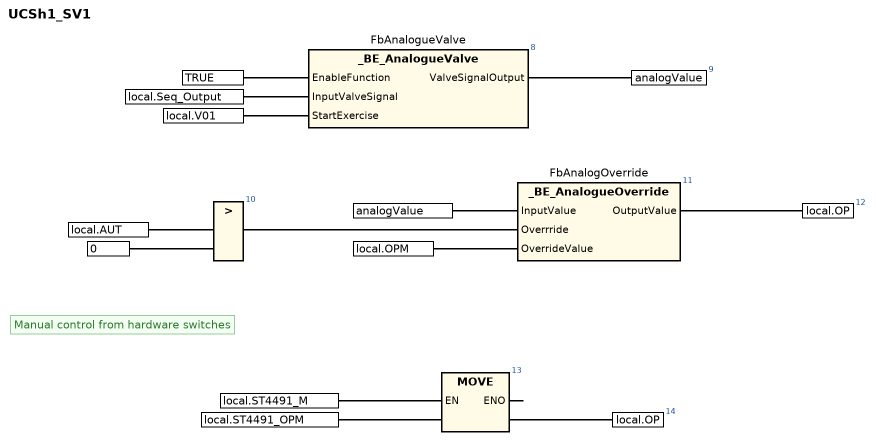
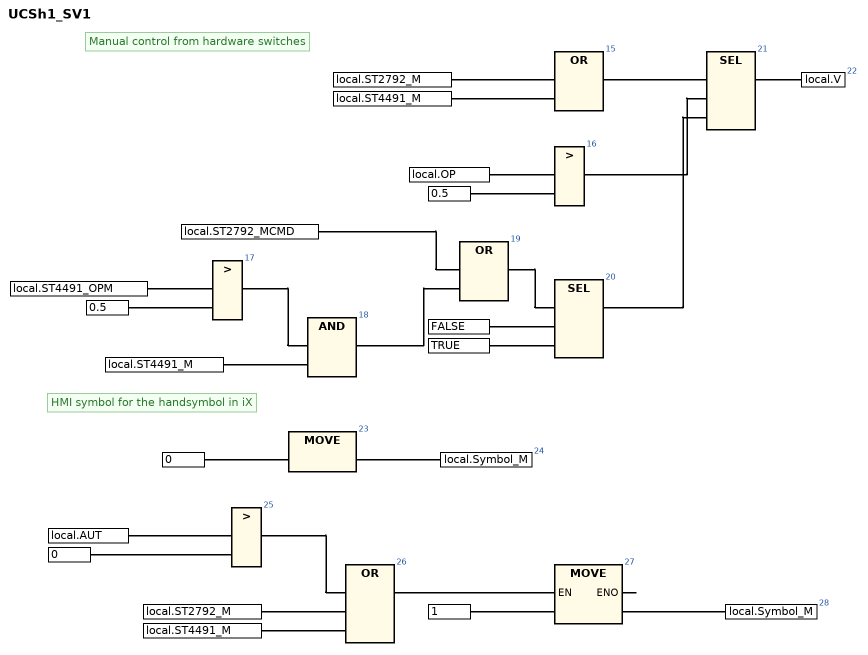
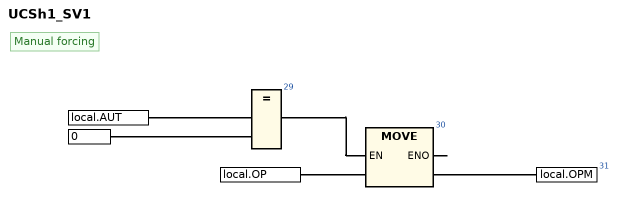
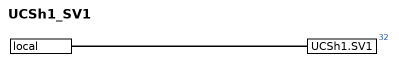
UCSh1.SV1.Seq_Output := UCSh1.GT1.OP;
local := UCSh1.SV1;
fbExercise(
    EnableFunction := local.Ex_En,
    RunIndication := local.OP > 0.5,
    DaysBetweenExercise := local.SP1,
    HoursBetweenExercise := local.SP2,
    EnableDay := local.Ex_En_Day,
    ExerciseStartDay := local.SP3,
    EnableHourMinute := local.Ex_En_Time,
    ExerciseStartHour := local.SP4,
    ExerciseStartMinute := local.SP5,
    ExerciseRunTime := local.SP6,
    SecondPulse := SYS_SecondPulse,
    ClockArray := SYS_ArrayPlcTime,
    SecondsIncObjectOff := local.Ex_SecOff,
    SavedWorkingData := local.Ex_SavedData); // _BE_Exercise
local.V01 := fbExercise.ExerciseActive;
local.PV1 := fbExercise.DaysLeft;
local.PV2 := fbExercise.HoursLeft;
local.PV3 := fbExercise.MinutesLeft;
FbAnalogueValve(EnableFunction := TRUE, InputValveSignal := local.Seq_Output, StartExercise := local.V01); // _BE_AnalogueValve
analogValue := FbAnalogueValve.ValveSignalOutput;
FbAnalogOverride(InputValue := analogValue, Overrride := local.AUT > 0, OverrideValue := local.OPM); // _BE_AnalogueOverride
local.OP := FbAnalogOverride.OutputValue;
// Manual control from hardware switches
IF local.ST4491_M THEN _w1 := local.ST4491_OPM; END_IF
local.OP := _w1;
// Manual control from hardware switches
local.V := SEL(local.ST2792_M OR local.ST4491_M, local.OP > 0.5, SEL(local.ST2792_MCMD OR local.ST4491_OPM > 0.5 AND local.ST4491_M, FALSE, TRUE));
// HMI symbol for the handsymbol in iX
local.Symbol_M := 0;
IF local.AUT > 0 OR local.ST2792_M OR local.ST4491_M THEN _w2 := 1; END_IF
local.Symbol_M := _w2;
// Manual forcing
IF local.AUT = 0 THEN _w3 := local.OP; END_IF
local.OPM := _w3;
UCSh1.SV1 := local;

END_PROGRAM

// Device/AREA1/System/SystemSignals/Sys_Version
PROGRAM Sys_Version
VAR
END_VAR

//POU handles version and date stamp in project.
//Version number
SYS_PLC_VersionNr:='1.00';

//Date stamp
SYS_PLC_VersionDate:='2014-12-18';

END_PROGRAM

// Device/AREA1/IO/Input/AnalogInput
PROGRAM AnalogInput
VAR
	scale_AI_1: _BE_ScaleAI8;
END_VAR
VAR // added by the converter: edge detectors and wires of the graphical bodies
    _w1 : ANY;
END_VAR

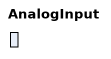
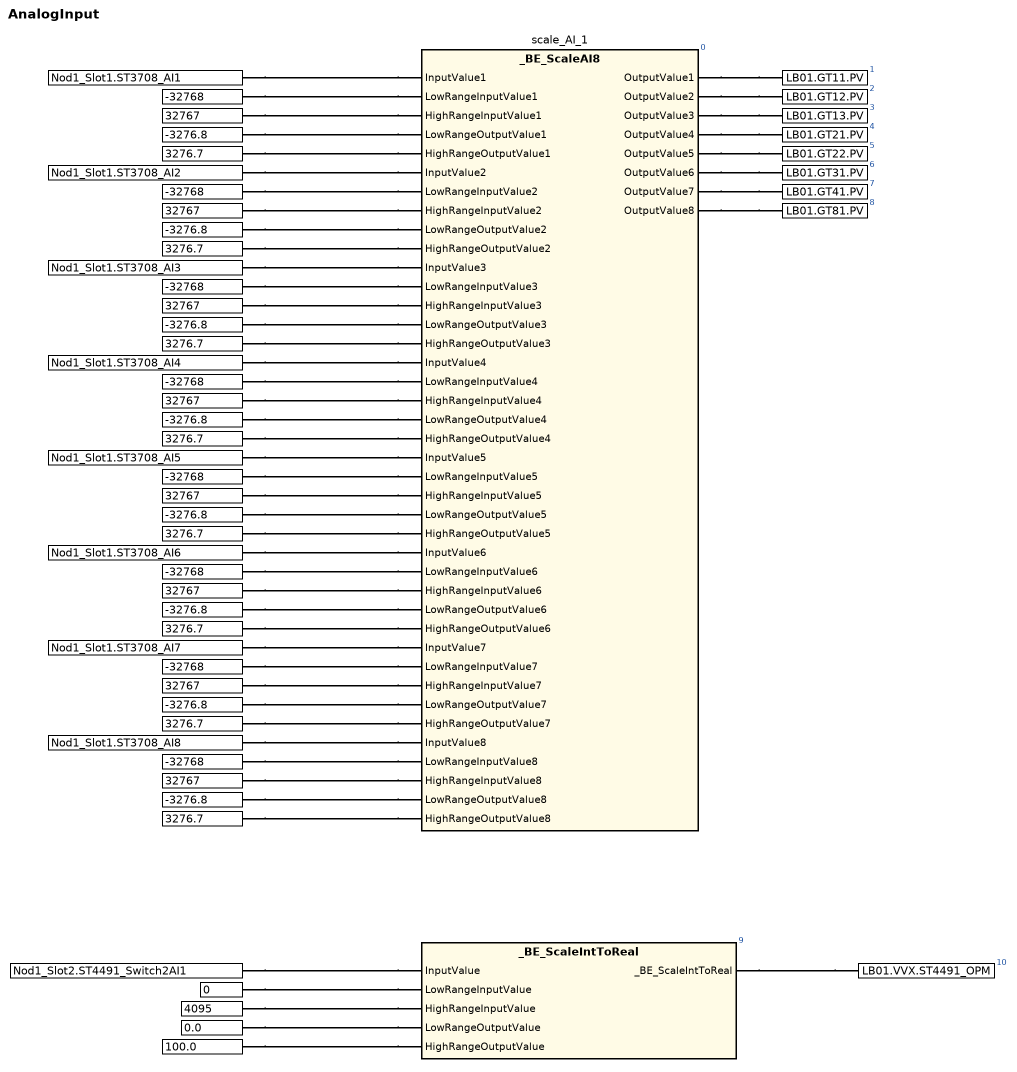
scale_AI_1(
    InputValue1 := Nod1_Slot1.ST3708_AI1,
    LowRangeInputValue1 := -32768,
    HighRangeInputValue1 := 32767,
    LowRangeOutputValue1 := -3276.8,
    HighRangeOutputValue1 := 3276.7,
    InputValue2 := Nod1_Slot1.ST3708_AI2,
    LowRangeInputValue2 := -32768,
    HighRangeInputValue2 := 32767,
    LowRangeOutputValue2 := -3276.8,
    HighRangeOutputValue2 := 3276.7,
    InputValue3 := Nod1_Slot1.ST3708_AI3,
    LowRangeInputValue3 := -32768,
    HighRangeInputValue3 := 32767,
    LowRangeOutputValue3 := -3276.8,
    HighRangeOutputValue3 := 3276.7,
    InputValue4 := Nod1_Slot1.ST3708_AI4,
    LowRangeInputValue4 := -32768,
    HighRangeInputValue4 := 32767,
    LowRangeOutputValue4 := -3276.8,
    HighRangeOutputValue4 := 3276.7,
    InputValue5 := Nod1_Slot1.ST3708_AI5,
    LowRangeInputValue5 := -32768,
    HighRangeInputValue5 := 32767,
    LowRangeOutputValue5 := -3276.8,
    HighRangeOutputValue5 := 3276.7,
    InputValue6 := Nod1_Slot1.ST3708_AI6,
    LowRangeInputValue6 := -32768,
    HighRangeInputValue6 := 32767,
    LowRangeOutputValue6 := -3276.8,
    HighRangeOutputValue6 := 3276.7,
    InputValue7 := Nod1_Slot1.ST3708_AI7,
    LowRangeInputValue7 := -32768,
    HighRangeInputValue7 := 32767,
    LowRangeOutputValue7 := -3276.8,
    HighRangeOutputValue7 := 3276.7,
    InputValue8 := Nod1_Slot1.ST3708_AI8,
    LowRangeInputValue8 := -32768,
    HighRangeInputValue8 := 32767,
    LowRangeOutputValue8 := -3276.8,
    HighRangeOutputValue8 := 3276.7); // _BE_ScaleAI8
LB01.GT11.PV := scale_AI_1.OutputValue1;
LB01.GT12.PV := scale_AI_1.OutputValue2;
LB01.GT13.PV := scale_AI_1.OutputValue3;
LB01.GT21.PV := scale_AI_1.OutputValue4;
LB01.GT22.PV := scale_AI_1.OutputValue5;
LB01.GT31.PV := scale_AI_1.OutputValue6;
LB01.GT41.PV := scale_AI_1.OutputValue7;
LB01.GT81.PV := scale_AI_1.OutputValue8;
_w1 := _BE_ScaleIntToReal(InputValue := Nod1_Slot2.ST4491_Switch2AI1, LowRangeInputValue := 0, HighRangeInputValue := 4095, LowRangeOutputValue := 0.0, HighRangeOutputValue := 100.0);
LB01.VVX.ST4491_OPM := _w1;

END_PROGRAM

// Device/AREA1/IO/Input/DigitalInput
PROGRAM DigitalInput
VAR
END_VAR

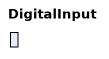
LB01.P1.V := Nod1_Slot3.strST1218;
LB01.P2.V := Nod1_Slot3.ST1218_DI1;
LB01.TF1.V := Nod1_Slot3.ST1218_DI2;
LB01.FF1.V := Nod1_Slot3.ST1218_DI3;
LB01.FireAlarm := Nod1_Slot3.ST1218_DI4;
LB01.GS91.InputAlarm := Nod1_Slot3.ST1218_DI5;
LB01.Overtime.CMD := Nod1_Slot3.ST1218_DI6;
LB01.GS91.InputAlarm := Nod1_Slot3.ST1218_DI7;
LB01.VVX.ST4491_M := Nod1_Slot2.ST4491_Switch1DI1;
LB01.TF1.ST2792_M := Nod1_Slot4.ST2792_Switch1DI1;
LB01.TF1.ST2792_MCMD := Nod1_Slot4.ST2792_Switch1DI2;
LB01.FF1.ST2792_M := Nod1_Slot4.ST2792_Switch2DI1;
LB01.FF1.ST2792_MCMD := Nod1_Slot4.ST2792_Switch2DI2;

END_PROGRAM

// Device/AREA1/IO/Output/AnalogOutput
PROGRAM AnalogOutput
VAR
	scale_AO_1: _BE_ScaleAO2;
END_VAR
VAR // added by the converter: edge detectors and wires of the graphical bodies
    _w1 : ANY;
END_VAR

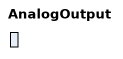
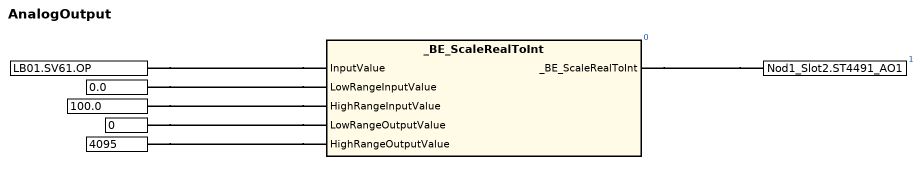
_w1 := _BE_ScaleRealToInt(InputValue := LB01.SV61.OP, LowRangeInputValue := 0.0, HighRangeInputValue := 100.0, LowRangeOutputValue := 0, HighRangeOutputValue := 4095);
Nod1_Slot2.ST4491_AO1 := _w1;

END_PROGRAM

// Device/AREA1/IO/Output/DigitalOutput
PROGRAM DigitalOutput
VAR
END_VAR

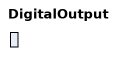
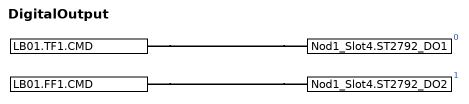
Nod1_Slot4.ST2792_DO1 := LB01.TF1.CMD;
Nod1_Slot4.ST2792_DO2 := LB01.FF1.CMD;

END_PROGRAM

// Device/AREA1/B001/LB01/Fan/FF1/LB01_FF1_OneSpeed
PROGRAM LB01_FF1_OneSpeed
VAR
	local:strFan_Onespeed;
	_BE_Fan2:_BE_Fan_2;
	AlarmFbAl01: _BE_AlarmAckRequired;
	AlarmFbAl02: _BE_AlarmAckRequired;
	fb_OperationalTime: _BE_OperationalTime;
	ackAl01: BOOL;
	ackAl02: BOOL;
	fanGuardOk: BOOL;
END_VAR

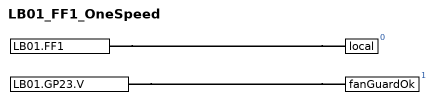
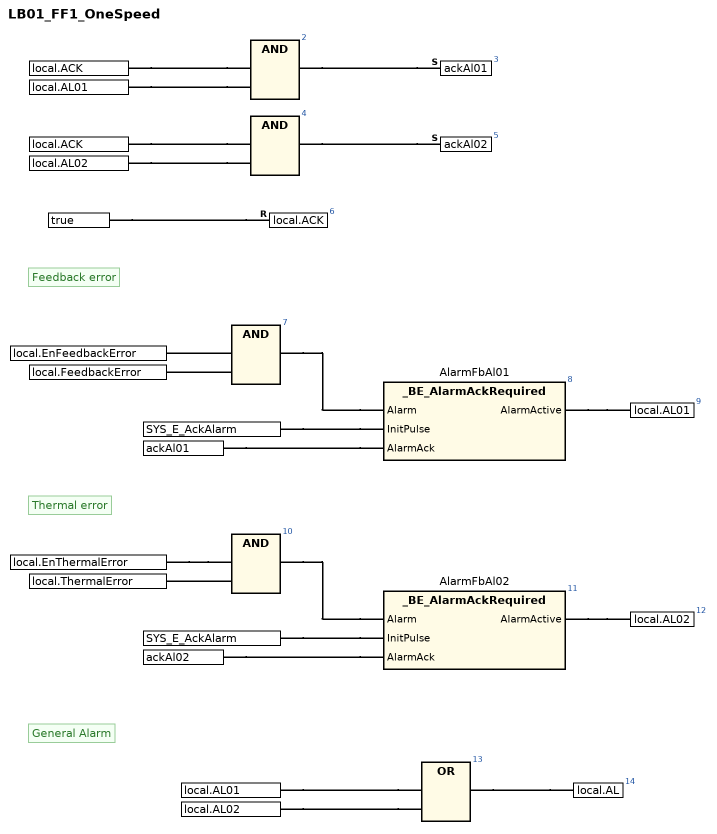
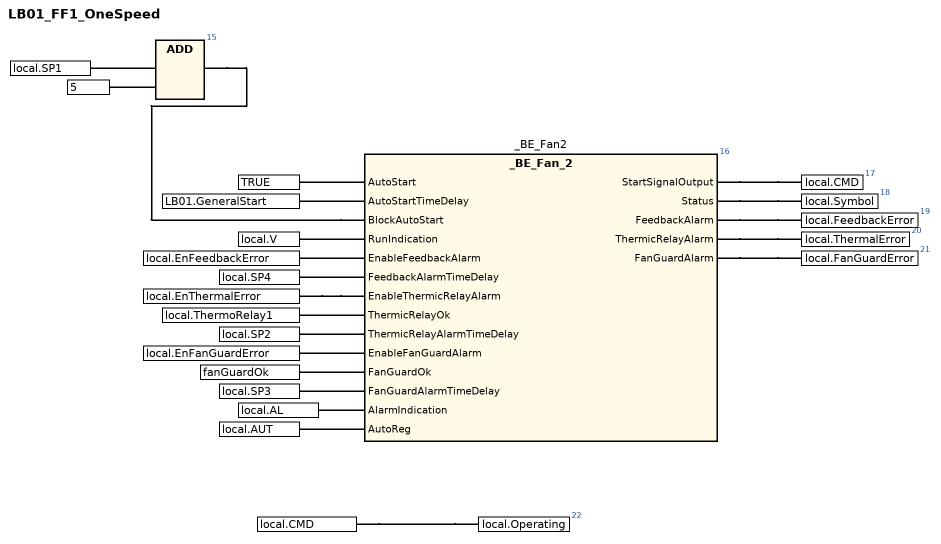
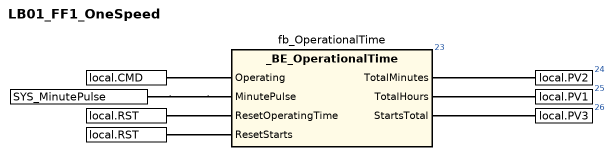
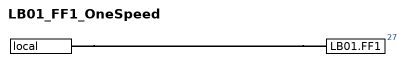
local := LB01.FF1;
fanGuardOk := LB01.GP23.V;
ackAl01 S= local.ACK AND local.AL01;
ackAl02 S= local.ACK AND local.AL02;
local.ACK R= true;
// Feedback error
AlarmFbAl01(
    Alarm := local.EnFeedbackError AND local.FeedbackError,
    InitPulse := SYS_E_AckAlarm,
    AlarmAck := ackAl01); // _BE_AlarmAckRequired
local.AL01 := AlarmFbAl01.AlarmActive;
// Thermal error
AlarmFbAl02(
    Alarm := local.EnThermalError AND local.ThermalError,
    InitPulse := SYS_E_AckAlarm,
    AlarmAck := ackAl02); // _BE_AlarmAckRequired
local.AL02 := AlarmFbAl02.AlarmActive;
// General Alarm
local.AL := local.AL01 OR local.AL02;
_BE_Fan2(
    AutoStart := TRUE,
    AutoStartTimeDelay := LB01.GeneralStart,
    BlockAutoStart := local.SP1 + 5,
    RunIndication := local.V,
    EnableFeedbackAlarm := local.EnFeedbackError,
    FeedbackAlarmTimeDelay := local.SP4,
    EnableThermicRelayAlarm := local.EnThermalError,
    ThermicRelayOk := local.ThermoRelay1,
    ThermicRelayAlarmTimeDelay := local.SP2,
    EnableFanGuardAlarm := local.EnFanGuardError,
    FanGuardOk := fanGuardOk,
    FanGuardAlarmTimeDelay := local.SP3,
    AlarmIndication := local.AL,
    AutoReg := local.AUT); // _BE_Fan_2
local.CMD := _BE_Fan2.StartSignalOutput;
local.Symbol := _BE_Fan2.Status;
local.FeedbackError := _BE_Fan2.FeedbackAlarm;
local.ThermalError := _BE_Fan2.ThermicRelayAlarm;
local.FanGuardError := _BE_Fan2.FanGuardAlarm;
local.Operating := local.CMD;
fb_OperationalTime(
    Operating := local.CMD,
    MinutePulse := SYS_MinutePulse,
    ResetOperatingTime := local.RST,
    ResetStarts := local.RST); // _BE_OperationalTime
local.PV2 := fb_OperationalTime.TotalMinutes;
local.PV1 := fb_OperationalTime.TotalHours;
local.PV3 := fb_OperationalTime.StartsTotal;
LB01.FF1 := local;

END_PROGRAM

// Device/AREA1/B001/LB01/Fan/FF1/LB01_FF1_TwoSpeed
PROGRAM LB01_FF1_TwoSpeed
VAR
	local:strFan_TwoSpeed;
	ControlTwoSpeed: _BE_FanTwoSpeed;
	AlarmFbAl03: _BE_AlarmAckRequired;
	AlarmFbAl04: _BE_AlarmAckRequired;
	AlarmFbAl05: _BE_AlarmAckRequired;
	AlarmFbAl06: _BE_AlarmAckRequired;
	ackAl03: BOOL;
	ackAl04: BOOL;
	ackAl05: BOOL;
	ackAl06: BOOL;
	fb_OperationalTime: _BE_OperationalTime;
	localV1: BOOL;
	localthermoRelay2: BOOL;
	fanGuardOk: BOOL;
END_VAR

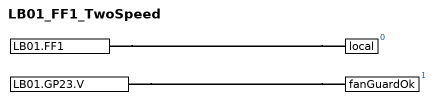
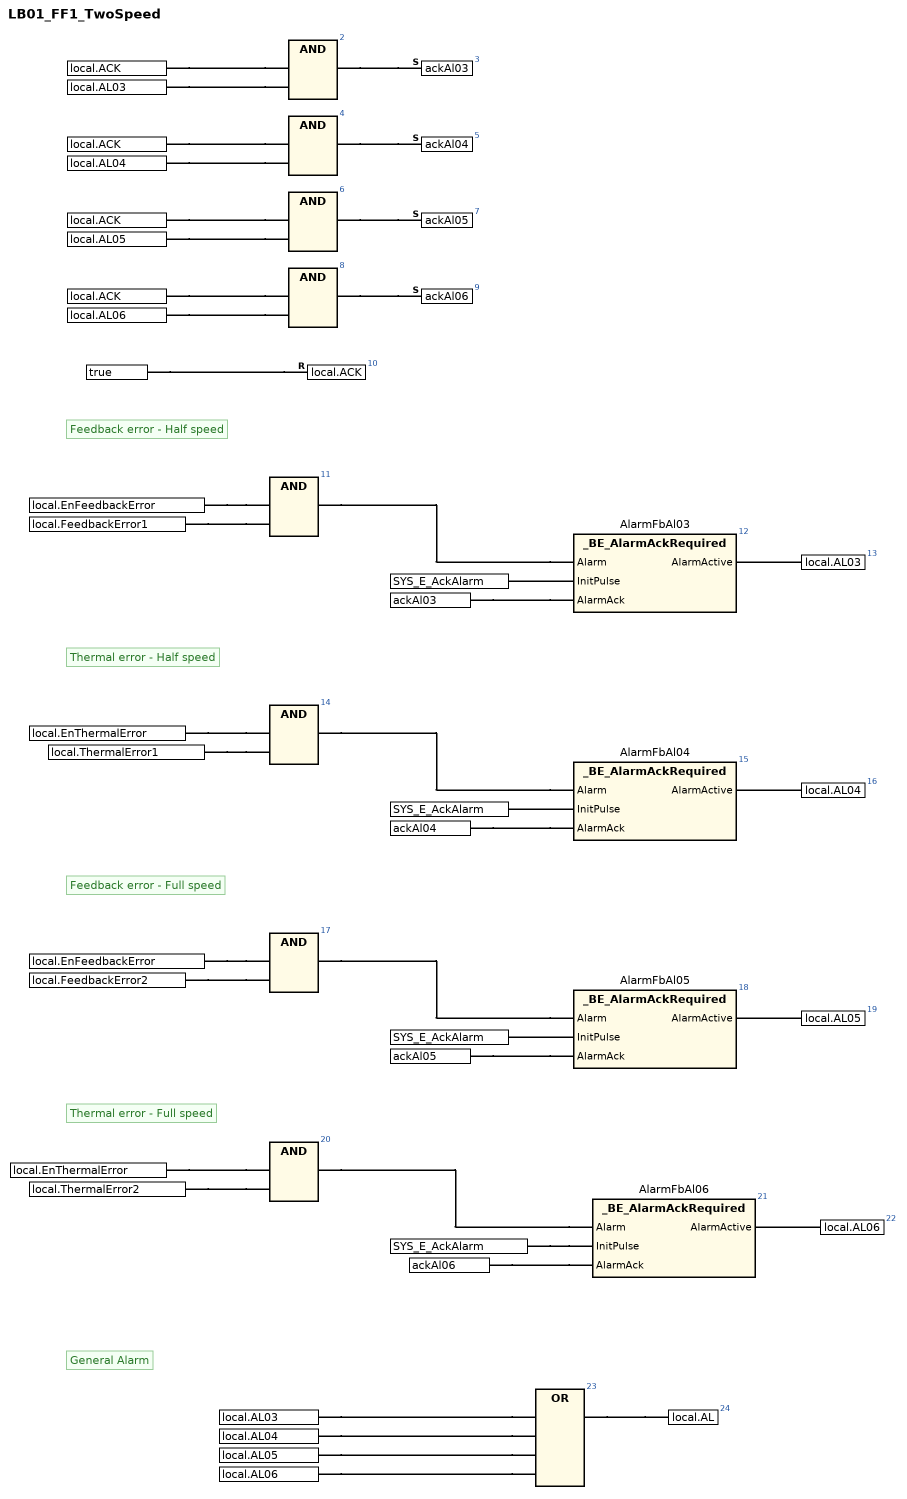
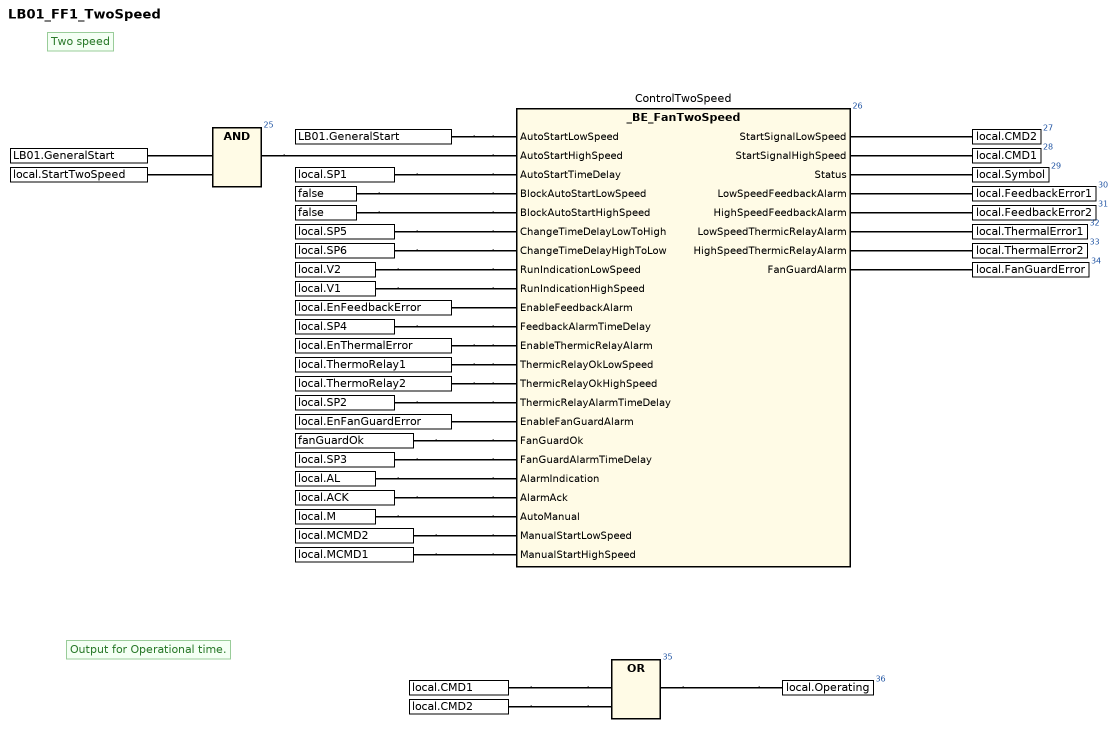
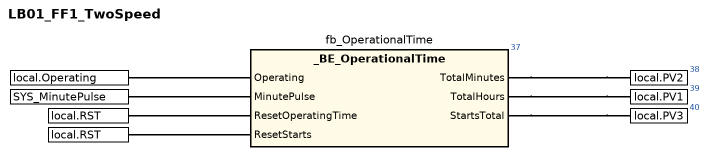
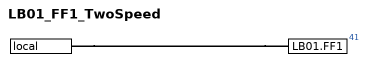
local := LB01.FF1;
fanGuardOk := LB01.GP23.V;
ackAl03 S= local.ACK AND local.AL03;
ackAl04 S= local.ACK AND local.AL04;
ackAl05 S= local.ACK AND local.AL05;
ackAl06 S= local.ACK AND local.AL06;
local.ACK R= true;
// Feedback error - Half speed
AlarmFbAl03(
    Alarm := local.EnFeedbackError AND local.FeedbackError1,
    InitPulse := SYS_E_AckAlarm,
    AlarmAck := ackAl03); // _BE_AlarmAckRequired
local.AL03 := AlarmFbAl03.AlarmActive;
// Thermal error - Half speed
AlarmFbAl04(
    Alarm := local.EnThermalError AND local.ThermalError1,
    InitPulse := SYS_E_AckAlarm,
    AlarmAck := ackAl04); // _BE_AlarmAckRequired
local.AL04 := AlarmFbAl04.AlarmActive;
// Feedback error - Full speed
AlarmFbAl05(
    Alarm := local.EnFeedbackError AND local.FeedbackError2,
    InitPulse := SYS_E_AckAlarm,
    AlarmAck := ackAl05); // _BE_AlarmAckRequired
local.AL05 := AlarmFbAl05.AlarmActive;
// Thermal error - Full speed
AlarmFbAl06(
    Alarm := local.EnThermalError AND local.ThermalError2,
    InitPulse := SYS_E_AckAlarm,
    AlarmAck := ackAl06); // _BE_AlarmAckRequired
local.AL06 := AlarmFbAl06.AlarmActive;
// General Alarm
local.AL := local.AL03 OR local.AL04 OR local.AL05 OR local.AL06;
// Two speed
ControlTwoSpeed(
    AutoStartLowSpeed := LB01.GeneralStart,
    AutoStartHighSpeed := LB01.GeneralStart AND local.StartTwoSpeed,
    AutoStartTimeDelay := local.SP1,
    BlockAutoStartLowSpeed := false,
    BlockAutoStartHighSpeed := false,
    ChangeTimeDelayLowToHigh := local.SP5,
    ChangeTimeDelayHighToLow := local.SP6,
    RunIndicationLowSpeed := local.V2,
    RunIndicationHighSpeed := local.V1,
    EnableFeedbackAlarm := local.EnFeedbackError,
    FeedbackAlarmTimeDelay := local.SP4,
    EnableThermicRelayAlarm := local.EnThermalError,
    ThermicRelayOkLowSpeed := local.ThermoRelay1,
    ThermicRelayOkHighSpeed := local.ThermoRelay2,
    ThermicRelayAlarmTimeDelay := local.SP2,
    EnableFanGuardAlarm := local.EnFanGuardError,
    FanGuardOk := fanGuardOk,
    FanGuardAlarmTimeDelay := local.SP3,
    AlarmIndication := local.AL,
    AlarmAck := local.ACK,
    AutoManual := local.M,
    ManualStartLowSpeed := local.MCMD2,
    ManualStartHighSpeed := local.MCMD1); // _BE_FanTwoSpeed
local.CMD2 := ControlTwoSpeed.StartSignalLowSpeed;
local.CMD1 := ControlTwoSpeed.StartSignalHighSpeed;
local.Symbol := ControlTwoSpeed.Status;
local.FeedbackError1 := ControlTwoSpeed.LowSpeedFeedbackAlarm;
local.FeedbackError2 := ControlTwoSpeed.HighSpeedFeedbackAlarm;
local.ThermalError1 := ControlTwoSpeed.LowSpeedThermicRelayAlarm;
local.ThermalError2 := ControlTwoSpeed.HighSpeedThermicRelayAlarm;
local.FanGuardError := ControlTwoSpeed.FanGuardAlarm;
// Output for Operational time.
local.Operating := local.CMD1 OR local.CMD2;
fb_OperationalTime(
    Operating := local.Operating,
    MinutePulse := SYS_MinutePulse,
    ResetOperatingTime := local.RST,
    ResetStarts := local.RST); // _BE_OperationalTime
local.PV2 := fb_OperationalTime.TotalMinutes;
local.PV1 := fb_OperationalTime.TotalHours;
local.PV3 := fb_OperationalTime.StartsTotal;
LB01.FF1 := local;

END_PROGRAM

// Device/AREA1/B001/LB01/Sensor/Temperature/GT31/LB01_GT31
PROGRAM LB01_GT31
VAR
	local:strSensor1;
	gt_Min: TON;
	gt_Max: TON;
	ackFault: BOOL;
	ackLal: BOOL;
	ackHal: BOOL;
	AlarmAcknowledge01: _BE_AlarmAckRemote;
	AlarmAcknowledge02: _BE_AlarmAckRemote;
	AlarmAcknowledge03: _BE_AlarmAckRemote;
END_VAR
VAR // added by the converter: edge detectors and wires of the graphical bodies
    _w1, _w3, _w4 : ANY;
    _w2 : BOOL;
END_VAR

